// TIA Portal V19 export
FUNCTION_BLOCK "Gestion"   // FB2, LAD
   VAR
      "Code erreur" : Word;
      "FM Noires" : Bool;
      "FM Mauvaises" : Bool;
      "FM Bonnes" : Bool;
   END_VAR
   VAR_TEMP   // added for the SCL form of the ladder/FBD networks
      _w1 : Bool;
   END_VAR
BEGIN

REGION Network 1: Scale de la valeur d'entrée analogique
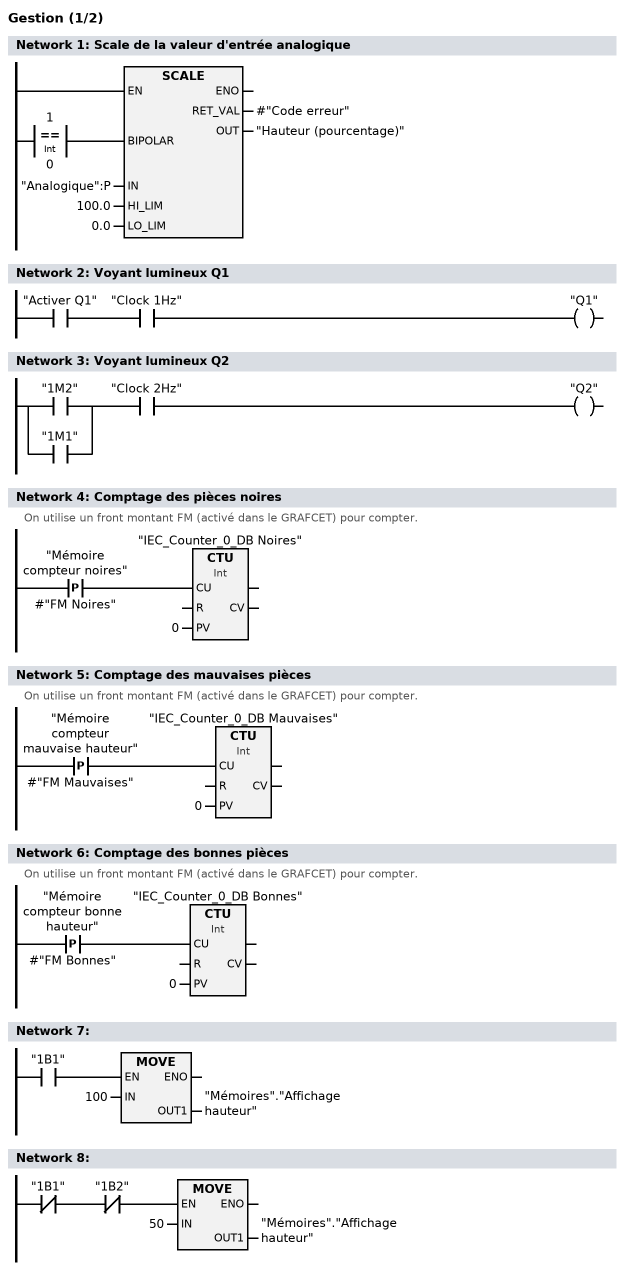
   #"Code erreur" := SCALE(BIPOLAR := 1 = 0,
                           IN := "Analogique":P,
                           HI_LIM := 100.0,
                           LO_LIM := 0.0,
                           OUT => "Hauteur (pourcentage)");
END_REGION

REGION Network 2: Voyant lumineux Q1
   RUNG wire#powerrail
      Contact( "Activer Q1" )
      Contact( "Clock 1Hz" )
      Coil( "Q1" )
   END_RUNG
   // the same network as SCL:
   "Q1" := "Activer Q1" AND "Clock 1Hz";
END_REGION

REGION Network 3: Voyant lumineux Q2
   RUNG wire#powerrail
      Contact( "1M2" )
      wire#w1
      Contact( "Clock 2Hz" )
      Coil( "Q2" )
   END_RUNG
   RUNG wire#powerrail
      Contact( "1M1" )
   END_RUNG wire#w1
   // the same network as SCL:
   "Q2" := ("1M2" OR "1M1") AND "Clock 2Hz";
END_REGION

REGION Network 4: Comptage des pièces noires
   // On utilise un front montant FM (activé dans le GRAFCET) pour compter.
   RUNG wire#powerrail
      P_Contact(operand := "Mémoire compteur noires", bit := #"FM Noires")
      { S7_Templates := "value_type := Int" } "IEC_Counter_0_DB Noires".CTU(r :=, pv := 0, cv =>)
   END_RUNG
   // the same network as SCL:
   #_w1 := "Mémoire compteur noires" AND NOT #"FM Noires";   // rising edge of "Mémoire compteur noires"
   #"FM Noires" := "Mémoire compteur noires";
   "IEC_Counter_0_DB Noires".CTU(CU := #_w1, PV := 0);
END_REGION

REGION Network 5: Comptage des mauvaises pièces
   // On utilise un front montant FM (activé dans le GRAFCET) pour compter.
   RUNG wire#powerrail
      P_Contact(operand := "Mémoire compteur mauvaise hauteur", bit := #"FM Mauvaises")
      { S7_Templates := "value_type := Int" } "IEC_Counter_0_DB Mauvaises".CTU(r :=, pv := 0, cv =>)
   END_RUNG
   // the same network as SCL:
   #_w1 := "Mémoire compteur mauvaise hauteur" AND NOT #"FM Mauvaises";   // rising edge of "Mémoire compteur mauvaise hauteur"
   #"FM Mauvaises" := "Mémoire compteur mauvaise hauteur";
   "IEC_Counter_0_DB Mauvaises".CTU(CU := #_w1, PV := 0);
END_REGION

REGION Network 6: Comptage des bonnes pièces
   // On utilise un front montant FM (activé dans le GRAFCET) pour compter.
   RUNG wire#powerrail
      P_Contact(operand := "Mémoire compteur bonne hauteur", bit := #"FM Bonnes")
      { S7_Templates := "value_type := Int" } "IEC_Counter_0_DB Bonnes".CTU(r :=, pv := 0, cv =>)
   END_RUNG
   // the same network as SCL:
   #_w1 := "Mémoire compteur bonne hauteur" AND NOT #"FM Bonnes";   // rising edge of "Mémoire compteur bonne hauteur"
   #"FM Bonnes" := "Mémoire compteur bonne hauteur";
   "IEC_Counter_0_DB Bonnes".CTU(CU := #_w1, PV := 0);
END_REGION

REGION Network 7
   RUNG wire#powerrail
      Contact( "1B1" )
      { S7_GenerateENO := "TRUE" } Move(in := 100, out1 => "Mémoires"."Affichage hauteur")
   END_RUNG
   // the same network as SCL:
   IF "1B1" THEN "Mémoires"."Affichage hauteur" := 100; END_IF;
END_REGION

REGION Network 8
   RUNG wire#powerrail
      I_Contact( "1B1" )
      I_Contact( "1B2" )
      { S7_GenerateENO := "TRUE" } Move(in := 50, out1 => "Mémoires"."Affichage hauteur")
   END_RUNG
   // the same network as SCL:
   IF NOT "1B1" AND NOT "1B2" THEN "Mémoires"."Affichage hauteur" := 50; END_IF;
END_REGION

REGION Network 9
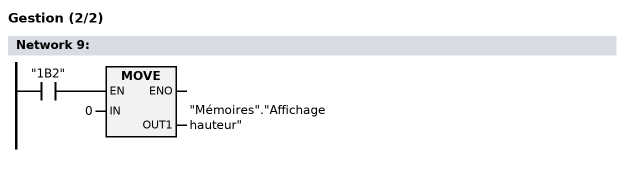
   RUNG wire#powerrail
      Contact( "1B2" )
      { S7_GenerateENO := "TRUE" } Move(in := 0, out1 => "Mémoires"."Affichage hauteur")
   END_RUNG
   // the same network as SCL:
   IF "1B2" THEN "Mémoires"."Affichage hauteur" := 0; END_IF;
END_REGION
END_FUNCTION_BLOCK
